FUNCTION FC_UnloadManager
VAR_IN_OUT
	UnloadingStation : BOOL;
	FLAGP : stByteAsBit;
END_VAR

UnloadingStation := TRUE;
IF FC_ProductStatus(FLAGP) <> eProductStatus.Scraped THEN
	FLAGP.aByte := 0;
	FLAGP.aBit.b0 := 1;
	FLAGP.aBit.b3 := 1;
END_IF

END_FUNCTION

(* stored: Version 1.1.0.1, ProductVersion 3.1.4024.15
   POU FC_UnloadManager: Id {fc94d719-39da-471c-8609-c5475ec7f060}, SpecialFunc None *)
